// TIA Portal V19 export
DATA_BLOCK "DB_JobData"   // DB3
{ S7_Optimized_Access := 'TRUE'; DB_Accessible_From_OPC_UA := 'FALSE' }
// stored: AutoNumber false, DBAccessibleFromOPCUA false, DBAccessibleFromWebserver false, MemoryReserve 100
   VAR RETAIN
      aJobData : Array[0..99] of "stJobData";   // Array of job data parameters
   END_VAR
BEGIN
END_DATA_BLOCK
